FUNCTION_BLOCK ABSTRACT TcoCylinderBase EXTENDS TcoCore.TcoComponent IMPLEMENTS ITcoCylinder
VAR_IN_OUT
	(*~
		<docu>
			<summary>
				Home position sensor.
			</summary>	
		</docu>
	~*)
	{attribute addProperty Name "<#Home position sensor#>"}
	inoAtHomePos : BOOL;
	(*~
		<docu>
			<summary>
				Working position sensor.
			</summary>	
		</docu>
	~*)
	{attribute addProperty Name "<#Work position sensor#>"}
	inoAtWorkPos : BOOL;
END_VAR
VAR_IN_OUT
	(*~
		<docu>
			<summary>
				Move to working home position signal.
			</summary>	
		</docu>
	~*)
	{attribute addProperty Name "<#Move to home position actuator#>"}
	inoToHomePos : BOOL;
	(*~
		<docu>
			<summary>
				Move to working posistion signal.
			</summary>	
		</docu>
	~*)
	{attribute addProperty Name "<#Move to work position actuator#>"}
	inoToWorkPos : BOOL;
END_VAR
VAR
	(*~
		<docu>
			<summary>
				Home position sensor.
			</summary>	
		</docu>
	~*)
	{attribute addProperty Name "<#Home position sensor#>"}
	_atHomePos : BOOL;
	(*~
		<docu>
			<summary>
				Working position sensor.
			</summary>	
		</docu>
	~*)
	{attribute addProperty Name "<#Work position sensor#>"}
	_atWorkPos : BOOL;
	(*~
		<docu>
			<summary>
				Move to working home position signal.
			</summary>	
		</docu>
	~*)
	{attribute addProperty Name "<#Move to home position actuator#>"}
	_toHomePos : BOOL;
	(*~
		<docu>
			<summary>
				Move to working posistion signal.
			</summary>	
		</docu>
	~*)
	{attribute addProperty Name "<#Move to work position actuator#>"}
	_toWorkPos : BOOL;
END_VAR

VAR
	{attribute addProperty Name "<#Home sensor signal#>"}
	_atHomePosSignalInfo : TcoCore.TcoSignalInfo;
	{attribute addProperty Name "<#Work sensor signal#>"}
    _atWorkPosSignalInfo : TcoCore.TcoSignalInfo;
	{attribute addProperty Name "<#Move to home position signal#>"}
    _toHomePosSignalInfo : TcoCore.TcoSignalInfo;
	{attribute addProperty Name "<#Move to work position signal#>"}
    _toWorkPosSignalInfo : TcoCore.TcoSignalInfo;
END_VAR

IF(__ISVALIDREF(inoAtHomePos)) THEN _atHomePos := inoAtHomePos; _atHomePosSignalInfo.GetSignalInfo(SIZEOF(inoAtHomePos), ADR(inoAtHomePos)); END_IF;
IF(__ISVALIDREF(inoAtWorkPos)) THEN _atWorkPos := inoAtWorkPos; _atWorkPosSignalInfo.GetSignalInfo(SIZEOF(inoAtWorkPos), ADR(inoAtWorkPos)); END_IF;
IF(__ISVALIDREF(inoToHomePos)) THEN inoToHomePos := _toHomePos; _toHomePosSignalInfo.GetSignalInfo(SIZEOF(inoToHomePos), ADR(inoToHomePos)); END_IF;
IF(__ISVALIDREF(inoToWorkPos)) THEN inoToWorkPos := _toWorkPos; _toWorkPosSignalInfo.GetSignalInfo(SIZEOF(inoToWorkPos), ADR(inoToWorkPos)); END_IF;

(*~
	<docu>
		<summary>
			Gets whether the piston is in home position. 		
		</summary>			
	</docu>	
~*)
PROPERTY AtHome : bool
GET
AtHome := THIS^._atHomePos;
END_GET
END_PROPERTY

(*~
	<docu>
		<summary>
			Gets whether the piston is in work position. 		
		</summary>			
	</docu>	
~*)
PROPERTY AtWork : bool
GET
AtWork := _atWorkPos;
END_GET
END_PROPERTY

METHOD FB_init : BOOL
VAR_INPUT
	bInitRetains : BOOL; // if TRUE, the retain variables are initialized (warm start / cold start)
	bInCopyCode : BOOL;  // if TRUE, the instance afterwards gets moved into the copy code (online change)
	ParentObject : ITcoObject;	
END_VAR
// This is not clear to me... I from time to time the consumer code does not see 'FB_init' of 'TcoObject', that's why overridden here with super call...
//SUPER^.FB_init(bInitRetains, bInCopyCode, ParentObject);
END_METHOD

(*~
	<docu>
		<summary>
			Gets the `MoveHomeTask` task that controls the moving of the cyclinder in home position.
			<remarks>			
				<note type="important">
					This is an abstract method and must be implemented in derived class.
				</note>
			</remarks>	 		
		</summary>			
	</docu>	
~*)
PROPERTY PUBLIC ABSTRACT MoveHomeTask : TcoCore.ITcoTask
GET
END_GET
END_PROPERTY

(*~
	<docu>
		<summary>
			Starts movement into home position. 		
		</summary>			
	</docu>	
~*)
METHOD MoveToHome : TcoCore.ITcoTaskStatus
IF(MoveHomeTask <> 0) THEN 
	MoveToHome := MoveHomeTask.Invoke();
END_IF;
END_METHOD

(*~
	<docu>
		<summary>
			Starts movement into work position. 		
		</summary>			
	</docu>	
~*)
METHOD MoveToWork :TcoCore.ITcoTaskStatus
IF(MoveWorkTask <> 0) THEN
	MoveToWork := MoveWorkTask.Invoke();
END_IF;
END_METHOD

(*~
	<docu>
		<summary>
			Gets the `MoveWorkTask` task that controls the moving of the cyclinder into work position.
			<remarks>			
				<note type="important">
					This is an abstract method and must be implemented in derived class.
				</note>
			</remarks>	 		
		</summary>			
	</docu>	
~*)
PROPERTY PUBLIC ABSTRACT MoveWorkTask : TcoCore.ITcoTask
GET
END_GET
END_PROPERTY

(*~
	<docu>
		<summary>
			Restore all tasks of this instance into initial state.		 		 		
		</summary>			
	</docu>	
~*)
METHOD  Restore : ITcoRestorable
IF(MoveHomeTask <> 0) THEN MoveHomeTask.Restore(); END_IF;
IF(MoveWorkTask <> 0) THEN MoveWorkTask.Restore(); END_IF;
IF(StopTask <> 0) THEN StopTask.Restore(); END_IF;
END_METHOD

METHOD PROTECTED  ServiceMode
END_METHOD

(*~
	<docu>
		<summary>
			Stops cyclinder movement.
		 	<remarks>			
				<note type="important">
					This method switched off the signals for the movement of the piston in both direction.
					However depending on the pnemumatics configuration the movement may contintue if designed in that way.
					THIS IS NOT A SAFETY FUCTION!
				</note>
			</remarks>	 		
		</summary>			
	</docu>	
~*)
METHOD Stop : TcoCore.ITcoTaskStatus
IF(StopTask <> 0) THEN
	Stop := StopTask.Invoke();
END_IF;
END_METHOD

(*~
	<docu>
		<summary>
			Gets the `StopTask` task that controls the stopping cyclinder movement.
			<remarks>			
				<note type="important">
					This is an abstract method and must be implemented in derived class.
				</note>
			</remarks>	 		
		</summary>			
	</docu>	
~*)
PROPERTY PUBLIC ABSTRACT StopTask : TcoCore.ITcoTask
GET
END_GET
END_PROPERTY

END_FUNCTION_BLOCK

(* stored: Version 1.1.0.1, ProductVersion 3.1.4024.9
   POU TcoCylinderBase: Id {3fb44fde-5170-065e-15db-1922ceae87e4}, SpecialFunc None
   Folder Operations: Id {29b1bf26-2e49-0157-2768-354cf52b72c1}
   Folder States: Id {8fae645c-458b-0e45-1bf7-768990103b17}
   Folder Tasks: Id {7be5fd98-9fb0-060c-1792-fcaa6c5bc4ff}
   Property AtHome: Id {5e107f57-e51c-0f79-3529-da3e4cb2b2bb}
   Get Get: Id {85dd945c-c8d1-02b7-0415-2a748f517767}
   Property AtWork: Id {dc8df1f9-093f-0f26-36a8-a4a685f63652}
   Get Get: Id {fe45a458-e620-0879-33f5-0609f376e566}
   Method FB_init: Id {bb291904-4fff-09da-220f-da3a28ae7cb5}
   Property MoveHomeTask: Id {fb0f0a8f-ab5f-0349-1e0f-f73ce363961c}
   Get Get: Id {88348909-5d81-0686-2b27-a47f3d3ade17}
   Method MoveToHome: Id {1bfcbfe1-eb41-0172-0520-bab3a7f92f43}
   Method MoveToWork: Id {e0e5e440-e0e8-0fa5-0117-09382853a221}
   Property MoveWorkTask: Id {590750ae-e716-0ddb-2979-6ad3642e47fb}
   Get Get: Id {3ed37472-e2ad-0855-245f-5291cb424419}
   Method Restore: Id {af413927-5e50-0360-15cc-4a40142811e3}
   Method ServiceMode: Id {52d34209-5bba-0f86-2d4c-15beb135d9d4}
   Method Stop: Id {aacfd4e0-4b15-025b-2310-d01828c9f71b}
   Property StopTask: Id {c0771b20-eee6-0635-3b50-f4038e2e02e3}
   Get Get: Id {ece7dc53-a76b-094f-1ea7-a013381f5c0b} *)
